(* IEC 61131-3 sources: IRIS-Project/LASAL CONTROL SOFTWARE/LasalProject_2025_09_25/Class/MPS, 1 file *)

(* ---- MPS.st ---- *)
(*!
<Class
	Name               = "MPS"
	Revision           = "0.0"
	RealtimeTask       = "false"
	CyclicTask         = "false"
	BackgroundTask     = "true"
	DefBackground      = "100 ms"
	Sigmatek           = "false"
	OSInterface        = "false"
	HighPriority       = "false"
	Automatic          = "false"
	UpdateMode         = "Prescan"
	SharedCommandTable = "true"
	Objectsize         = "(600,300)">
	<Channels>
		<Server Name="ClassSvr" Visualized="false" Initialize="false" WriteProtected="true" Retentive="false"/>
		<Server Name="Ok_From_MPS" Visualized="false" Initialize="false" WriteProtected="false" Retentive="false"/>
		<Server Name="ReqToMPS" Visualized="false" Initialize="false" WriteProtected="false" Retentive="false"/>
		<Server Name="s_MPS_ACK" Visualized="false" Initialize="false" WriteProtected="false" Retentive="false"/>
		<Client Name="ACKFromMPS" Required="true" Internal="false"/>
		<Client Name="c_ReqToMPS" Required="true" Internal="false"/>
		<Client Name="To_CameraAlignment_Power" Required="true" Internal="false"/>
		<Client Name="To_Manager_Motori" Required="true" Internal="false"/>
	</Channels>
</Class>
*)
MPS : CLASS
	TYPE
	  CaseMPS :  //! <Type Public="true" Name="CaseMPS"/>
	  (
	    MPS_Idle,
	    MPS_Ok_To_IRIS,
	    MPS_No_To_IRIS
	  )$UDINT;
	END_TYPE
  //Servers:
	ClassSvr 	: SvrChCmd_DINT;
	ReqToMPS 	: SvrCh_DINT;
	Ok_From_MPS 	: SvrCh_CaseMPS_PTofCls_MPS;
	s_MPS_ACK 	: SvrCh_DINT;
  //Clients:
	To_Manager_Motori 	: CltCh_DINT;
	ACKFromMPS 	: CltCh_DINT;
	c_ReqToMPS 	: CltCh_DINT;
	To_CameraAlignment_Power 	: CltCh_DINT;
  //Variables:
		v_CaseMPS 	: CaseMPS;
		ACK 	: DINT;
  //Functions:

	FUNCTION VIRTUAL GLOBAL Init;

	FUNCTION VIRTUAL GLOBAL Background
		VAR_INPUT
			EAX 	: UDINT;
		END_VAR
		VAR_OUTPUT
			state (EAX) 	: UDINT;
		END_VAR;

	FUNCTION VIRTUAL GLOBAL ReqToMPS::Read
		VAR_OUTPUT
			output (EAX) 	: DINT;
		END_VAR;
  //Tables:
	FUNCTION @STD
		VAR_OUTPUT
			ret_code	: CONFSTATES;
		END_VAR;
	FUNCTION GLOBAL TAB @CT_;
END_CLASS;

FUNCTION VIRTUAL GLOBAL MPS::Background
	VAR_INPUT
		EAX 	: UDINT;
	END_VAR
	VAR_OUTPUT
		state (EAX) 	: UDINT;
	END_VAR

  //ACK:=ACKFromMPS.Read(); -> da togliere il commento quando bisogna utilizzare l'ingresso fisico
  s_MPS_ACK.Write(input:=ACK);

  if ReqToMPS.Read() then
    c_ReqToMPS.Write(input:=1);
  else
    c_ReqToMPS.Write(input:=0);
  end_if;

  if ACK then
    v_CaseMPS:=MPS_Ok_To_IRIS;
  else
    v_CaseMPS:=MPS_No_To_IRIS;
  end_if;

  case v_CaseMPS of

  MPS_Idle:

  MPS_Ok_To_IRIS:

    To_Manager_Motori.Write(input:=1);
    To_CameraAlignment_Power.Write(input:=600);//scrivo 600 -> maxCurrent al modulo st151 associato a M6
  //NON DISCOMMENTARE  //Ok_From_MPS.Write(input:=MPS_No_To_IRIS);//faccio questo passaggio altrimenti nel Manager_Motori Rimane la variabile a 1

  MPS_No_To_IRIS:

    To_Manager_Motori.Write(input:=0);
   //NON DISCOMMENTARE //Ok_From_MPS.Write(input:=MPS_Idle);
    To_CameraAlignment_Power.Write(input:=0);//scrivo 0 -> maxCurrent al modulo st151 associato a M6
  end_case;

	state := READY;

END_FUNCTION

FUNCTION VIRTUAL GLOBAL MPS::ReqToMPS::Read
	VAR_OUTPUT
		output (EAX) 	: DINT;
	END_VAR

	output := ReqToMPS;

END_FUNCTION

FUNCTION VIRTUAL GLOBAL MPS::Init
ACK:=0;
END_FUNCTION
